// TIA Portal V16 export
// export: Created 2021-03-19T11:45:00.1547818Z, ExportSetting WithDefaults, DisplayName Totally Integrated Automation Portal, DisplayVersion V16 Update 3, DisplayName TIA Portal Version Control Interface, DisplayVersion V16 Update 2, DisplayName TIA Portal Openness, DisplayVersion V16 Update 3, DisplayName STEP 7 Professional, DisplayVersion V16 Update 3, DisplayName STEP 7 Safety, DisplayVersion V16, DisplayName WinCC Professional, DisplayVersion V16 Update 3
TYPE "UT21001_Dy_SysData"
TITLE = Dynamic UDT — Sys - Global Data
// Global System Data
// stored: IsFailsafeCompliant false
   STRUCT
      revInfo { ExternalWritable := 'False'} : "UT01000_St_SysRevision";   // ▀▀▀▀ UDT CURRENT REVISION
      ___________0010_0 { ExternalAccessible := 'False'; ExternalVisible := 'False'; ExternalWritable := 'False'} : Bool;
      ___________0010_1 { ExternalAccessible := 'False'; ExternalVisible := 'False'; ExternalWritable := 'False'} : Bool;   // ▀▀▀▀ CYCLE TIME DATA
      CycTime_Prev { ExternalWritable := 'False'} : Real;   // Previous cycle time (ms)
      CycTime_Max { ExternalWritable := 'False'} : Real;   // Maximum cycle time - since start-up (ms)
      CycTime_Min { ExternalWritable := 'False'} : Real;   // Minimum cycle time - since start-up (ms)
      Cyc_Counter { ExternalWritable := 'False'} : UDInt;   // Cycle rolling counter - incremented by 1 each scan
      __________0020_0 { ExternalAccessible := 'False'; ExternalVisible := 'False'; ExternalWritable := 'False'} : Bool := false;
      __________0020_1 { ExternalAccessible := 'False'; ExternalVisible := 'False'; ExternalWritable := 'False'} : Bool := false;   // ▀▀▀▀ REAL TIME CLOCK DATA
      RTC_Year { ExternalWritable := 'False'} : Int;   // Year (returns a value in the range 1970 to 2262)
      RTC_Month { ExternalWritable := 'False'} : Int;   // Month (1-12 representing Jan to Dec)
      RTC_Day { ExternalWritable := 'False'} : Int;   // Day of month (1-31)
      RTC_DayofWeek { ExternalWritable := 'False'} : Int;   // Day of week (1-7, where 1=Sunday, 7=Saturday)
      RTC_Hour { ExternalWritable := 'False'} : Int;   // Hour of day (0-23)
      RTC_Minute { ExternalWritable := 'False'} : Int;   // Minutes (0-59)
      RTC_Second { ExternalWritable := 'False'} : Int;   // Seconds (0-59)
      RTC_millisecond { ExternalWritable := 'False'} : Int;   // Milliseconds (0-999)
   END_STRUCT;
   // revInfo.REV_BLOCK := 'UT21001';
   // revInfo.REV_NUMBER := '001.000';
   // revInfo.REV_DATE := '2021-02-18';
   // revInfo.REV_AUTHOR := 'M. Gledhill ';
END_TYPE
